(*

.. <legal notes>

legal notes
=================
| SPDX-FileCopyrightText: © 2026 Oleksandr Tiutyk <trofimich@gmail.com>
| SPDX-License-Identifier: LGPL-3.0-only
| For details check: LGPL-3.0-only_

.. _LGPL-3.0-only: https://www.gnu.org/licenses/lgpl-3.0.en.html

.. </legal notes>

*)

PROGRAM SignedByteHelper
VAR CONSTANT
	MIN_VALUE : SINT := -128;
	MAX_VALUE : SINT := +127;
END_VAR
VAR
	_ClassName : STRING := __POUNAME();
END_VAR

{attribute 'monitoring' := 'call'}
PROPERTY ClassName : STRING
GET
ClassName := _ClassName;
END_GET
END_PROPERTY

{attribute 'monitoring' := 'call'}
PROPERTY NamespaceName : STRING
GET
NamespaceName := CurrentNamespace.Name;
END_GET
END_PROPERTY

END_PROGRAM

(* stored: Version 1.1.0.1
   POU SignedByteHelper: Id {7cacf48f-3d2a-40d3-b0ed-66de154a8a38}, SpecialFunc None
   Property ClassName: Id {1aecd1fc-e59b-425b-beb8-6a69d1203863}
   Get Get: Id {ef4d7596-1587-4aa9-b7e0-1b637dcd8aa9}
   Property NamespaceName: Id {fceddc2e-9224-43d3-8200-31540650f86f}
   Get Get: Id {92be5abe-c32f-441d-8d6e-c53b7aa2d651} *)
